// TwinCAT 3 PLC project Alarmbewaking
// ProgramVersion: 3.1.4024.0
// libraries:
//   Tc2_Standard, * (Beckhoff Automation GmbH)
//   Tc2_System, * (Beckhoff Automation GmbH)
//   Tc3_Module, * (Beckhoff Automation GmbH)
// project tree:
//   / PlcTask.TcTTO
//   POUs/ MAIN.TcPOU

CONFIGURATION Alarmbewaking
    RESOURCE PLC ON TwinCAT3
        TASK PlcTask(INTERVAL := T#10ms, PRIORITY := 25);
        PROGRAM MAIN WITH PlcTask : MAIN;
    END_RESOURCE
END_CONFIGURATION

// ---- POUs/MAIN.TcPOU
PROGRAM MAIN
VAR
	
// Inputs
	S01 AT %I*: BOOL; // Sensor 1
	S02 AT %I*: BOOL; // Sensor 2
	S03 AT %I*: BOOL; // Sensor 3

// Outputs
	L1 AT %Q*: BOOL; // Lamp 1
	L2 AT %Q*: BOOL; // Lamp 2
	L3 AT %Q*: BOOL; // Lamp 3
	L4 AT %Q*: BOOL; // Lamp 4
	L5 AT %Q*: BOOL; // Lamp 5
	Reset_DK AT %Q*: BOOL; // Reset Drukknop 1
	
END_VAR

(*
Alarmbewaking (6 regels code)

In een vat wordt een proces bewaakt met 3 sensoren

    Sensor1 meet de druk. TRUE bij een te hoge druk.
    Sensor2 meet de temperatuur. TRUE bij een te hoge temperatuur.
    Sensor3 meet het vloeistofniveau. FALSE bij een te laag niveau.

Er zijn 5 lampen die als indicator dienen voor het proces:

    Lamp1 gaat aan als de druk te hoog is.
    Lamp2 gaat aan als de temperatuur te hoog is.
    Lamp3 gaat aan als het niveau te laag is.
    Bovenstaande lampen gaan automatisch uit als er geen melding meer gegeven hoeft te worden.
	
    Lamp4 gaat aan als er zich twee alarmen gelijktijdig voordoen. 
	Van zodra er geen twee alarmen meer zijn gaat deze lamp uit. 
	Bij drie alarmen gaat deze lamp ook uit.
    Lamp5 gaat aan als er drie alarmen zijn. 
	Deze lamp blijft aan, ook nadat er geen drie alarmen meer zijn. 
	De lamp kan enkel uitgeschakeld worden met een extra drukknop.
*)

 
L1 := S01; // Drukalarm
L2 := S02; // Temperatuuralarm
L3 := NOT S03; // Niveau-Alarm
L4 := (S01 AND S02 AND NOT S03) OR (S01 AND NOT S02 AND S03) OR (NOT S01 AND S02 AND S03); // Twee alarmen
L5 := L5 OR (S01 AND S02 AND NOT S03); // Drie alarmen
IF Reset_DK THEN L5 := FALSE; END_IF; // Reset Lamp5 enkel met drukknop

END_PROGRAM
